{attribute 'pack_mode' := '1'}
TYPE ST_CalibDone EXTENDS ST_MsgToCCS:
STRUCT
    homePosition		: ARRAY [0..1] OF LREAL;
    deployedPosition	: ARRAY [0..1] OF LREAL;
    (* hallPosCal[a, d, t] is coordinate of
       the (t+1)st transition that occurred
       while moving axis a+1 in direction d.
       d=0 for positive, d=1 for negative.
     *)
    hallPosCal			: ARRAY [0..1, 0..1, 0..239] OF LREAL;
END_STRUCT
END_TYPE

(* stored: Version 1.1.0.1, ProductVersion 3.1.4024.3
   DUT ST_CalibDone: Id {ec263d66-2e57-4d76-8ae5-dc79b75b3e1c} *)
